PROGRAM MAIN
VAR
	xStart : BOOL := FALSE;
	xEStop : BOOL := FALSE; 
	xMotor : BOOL := FALSE;
	xEnable : BOOL := FALSE;
	XLocked : BOOL := FALSE;
	xInTimer : BOOL:= FALSE;
	fbTMR : TON;
END_VAR



xEnable := (xStart OR xEnable) AND NOT xEStop AND NOT xLocked;


IF xEStop THEN 
	
	xLocked := TRUE;
	xInTimer := TRUE;
	
END_IF

fbTMR(IN := xInTimer,
	PT := T#10S );
	

IF fbTMR.Q THEN
	
	xLocked := FALSE;
	xInTimer := FALSE;

END_IF

END_PROGRAM

(* stored: Version 1.1.0.1, ProductVersion 3.1.4024.11
   POU MAIN: Id {66339b33-5525-4df3-9b4e-ac5b6239f1e4}, SpecialFunc None *)
